// SIMATIC S7-200 project (STEP 7-Micro/WIN), CPU 224XP REL 02.01

SYMBOL_TABLE USER1
P0               M0.0
END_SYMBOL_TABLE

ORGANIZATION_BLOCK MAIN:OB1
TITLE=PROGRAM COMMENTS
BEGIN
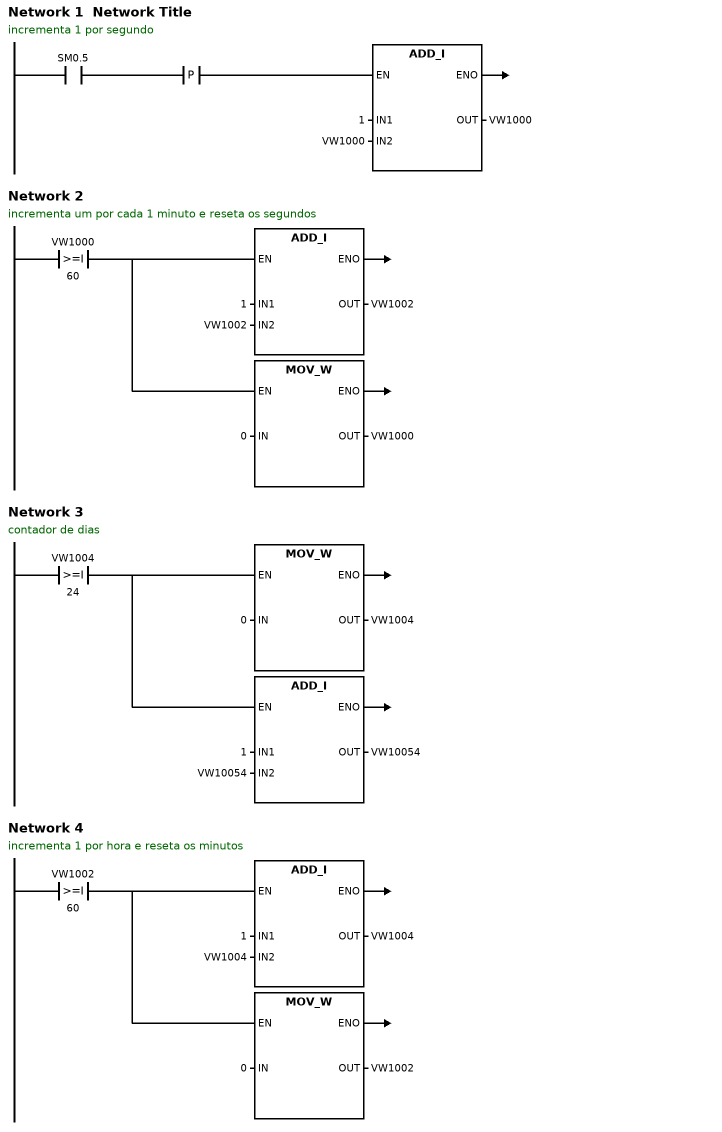
Network 1 // Network Title
// incrementa 1 por segundo
LD     SM0.5
EU
+I     1, VW1000
Network 2
// incrementa um por cada 1 minuto e reseta os segundos
LDW>=  VW1000, 60
+I     1, VW1002
MOVW   0, VW1000
Network 3
// contador de dias
LDW>=  VW1004, 24
MOVW   0, VW1004
+I     1, VW10054
Network 4
// incrementa 1 por hora e reseta os minutos
LDW>=  VW1002, 60
+I     1, VW1004
MOVW   0, VW1002
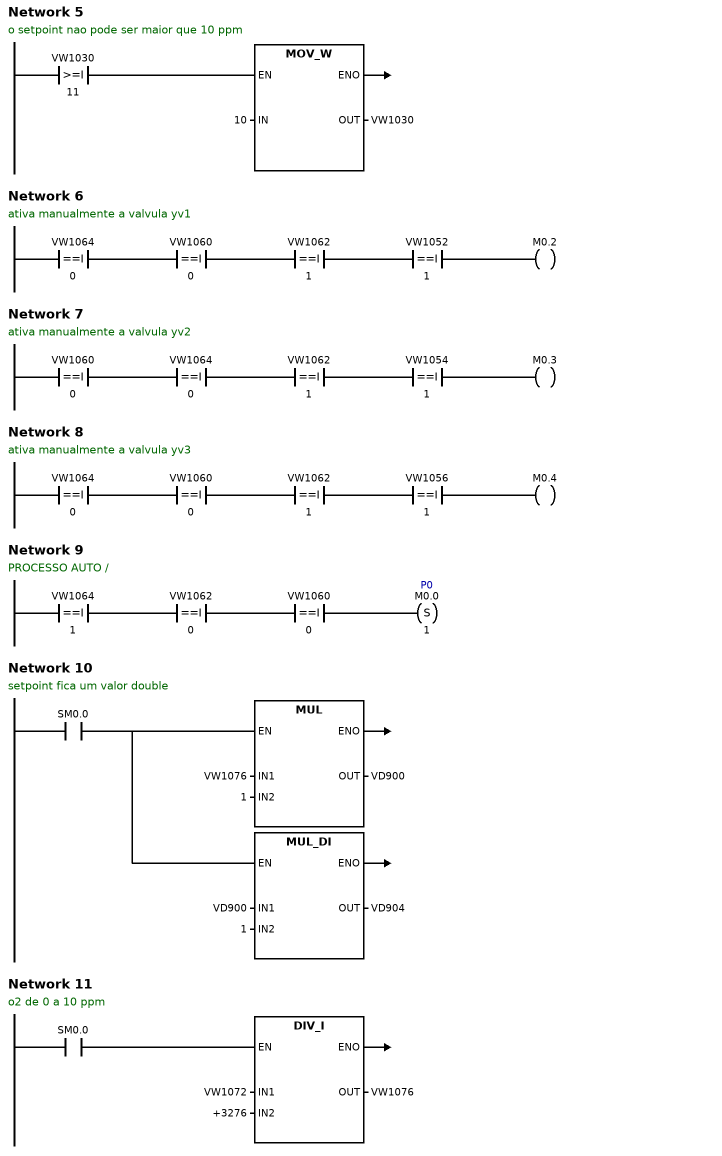
Network 5
// o setpoint nao pode ser maior que 10 ppm
LDW>=  VW1030, 11
MOVW   10, VW1030
Network 6
// ativa manualmente a valvula yv1
LDW=   VW1064, 0
AW=    VW1060, 0
AW=    VW1062, 1
AW=    VW1052, 1
=      M0.2
Network 7
// ativa manualmente a valvula yv2
LDW=   VW1060, 0
AW=    VW1064, 0
AW=    VW1062, 1
AW=    VW1054, 1
=      M0.3
Network 8
// ativa manualmente a valvula yv3
LDW=   VW1064, 0
AW=    VW1060, 0
AW=    VW1062, 1
AW=    VW1056, 1
=      M0.4
Network 9
// PROCESSO AUTO
// 
LDW=   VW1064, 1
AW=    VW1062, 0
AW=    VW1060, 0
S      P0:M0.0, 1
Network 10
// setpoint fica um valor double
LD     SM0.0
MOVW   VW1076, VW902
MUL    1, VD900
MOVD   VD900, VD904
*D     1, VD904
Network 11
// o2 de 0 a 10 ppm
LD     SM0.0
MOVW   VW1072, VW1076
/I     +3276, VW1076
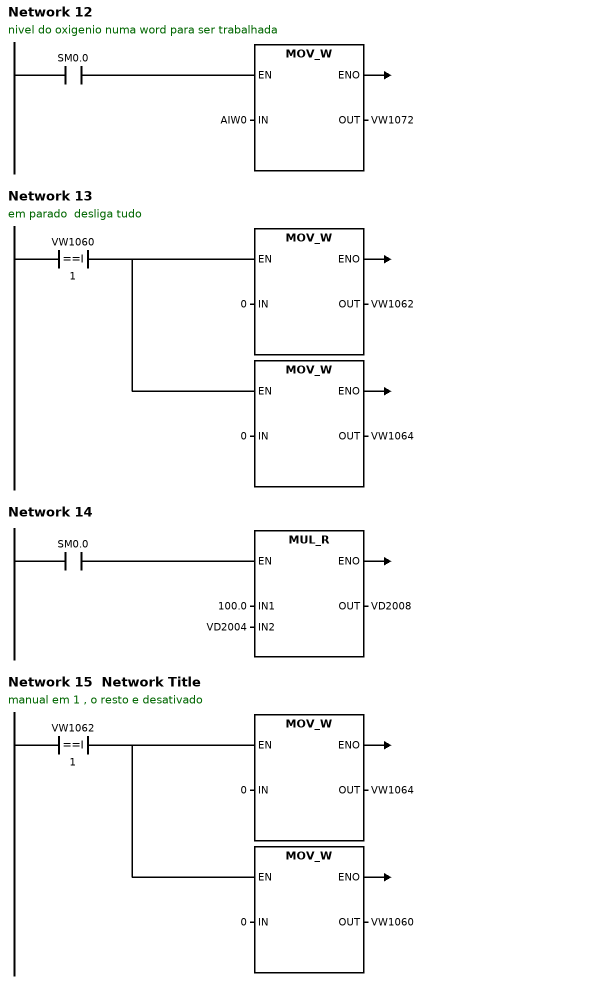
Network 12
// nivel do oxigenio numa word para ser trabalhada 
LD     SM0.0
MOVW   AIW0, VW1072
Network 13
// em parado  desliga tudo
LDW=   VW1060, 1
MOVW   0, VW1062
MOVW   0, VW1064
Network 14
LD     SM0.0
MOVR   100.0, VD2008
*R     VD2004, VD2008
Network 15 // Network Title
// manual em 1 , o resto e desativado
LDW=   VW1062, 1
MOVW   0, VW1064
MOVW   0, VW1060
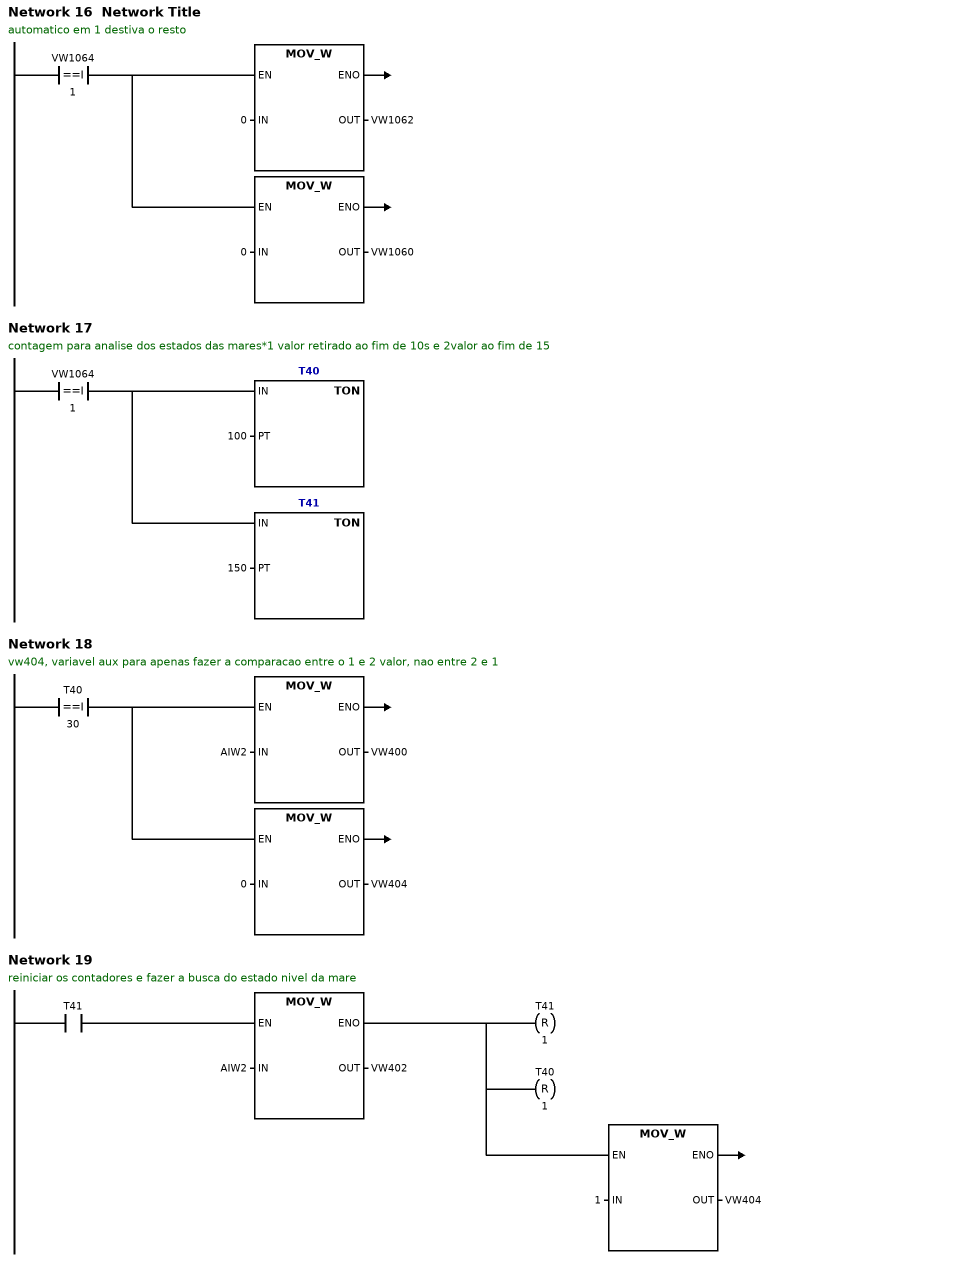
Network 16 // Network Title
// automatico em 1 destiva o resto
LDW=   VW1064, 1
MOVW   0, VW1062
MOVW   0, VW1060
Network 17
// contagem para analise dos estados das mares*1 valor retirado ao fim de 10s e 2valor ao fim de 15
LDW=   VW1064, 1
TON    T40, 100
TON    T41, 150
Network 18
// vw404, variavel aux para apenas fazer a comparacao entre o 1 e 2 valor, nao entre 2 e 1
LDW=   T40, 30
MOVW   AIW2, VW400
MOVW   0, VW404
Network 19
// reiniciar os contadores e fazer a busca do estado nivel da mare
LD     T41
MOVW   AIW2, VW402
AENO
R      T41, 1
R      T40, 1
MOVW   1, VW404
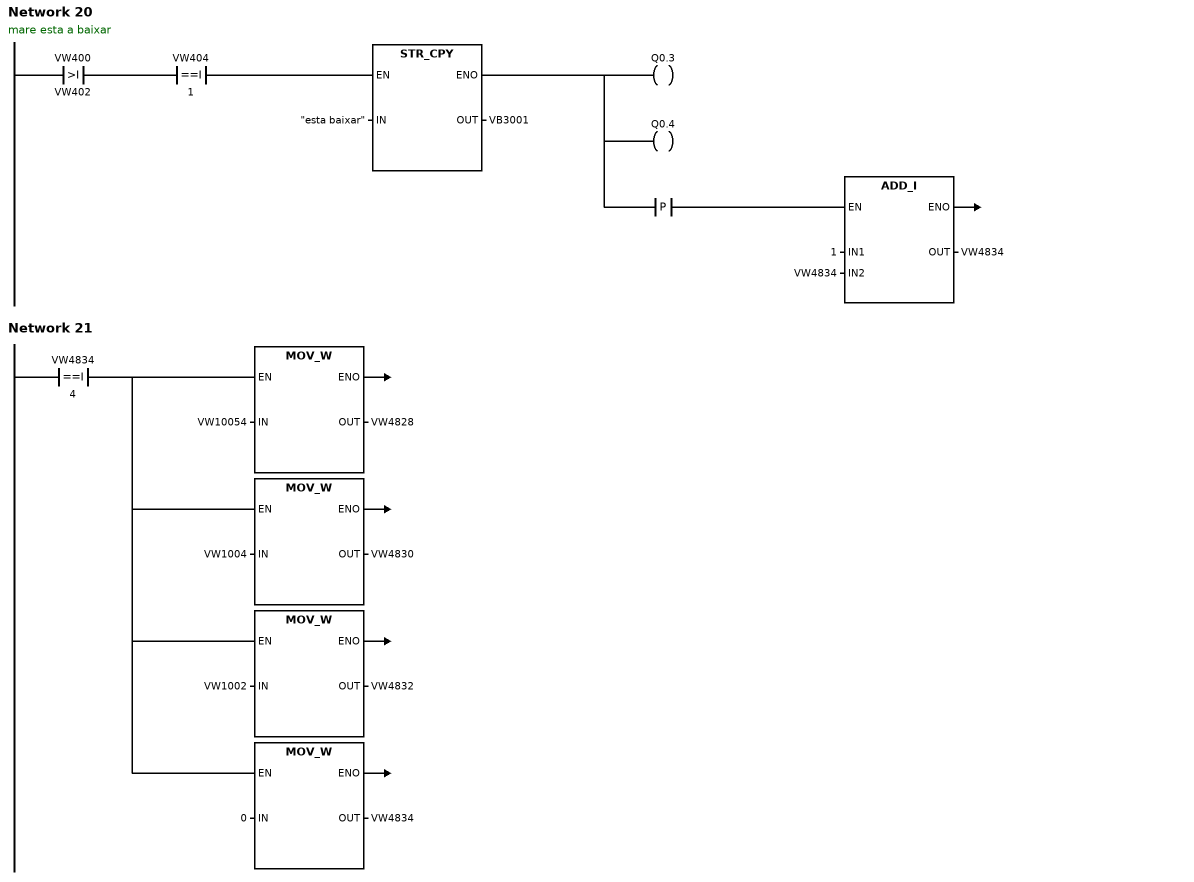
Network 20
// mare esta a baixar
LDW>   VW400, VW402
AW=    VW404, 1
SCPY   "esta baixar", VB3001
AENO
=      Q0.3
=      Q0.4
EU
+I     1, VW4834
Network 21
LDW=   VW4834, 4
MOVW   VW10054, VW4828
MOVW   VW1004, VW4830
MOVW   VW1002, VW4832
MOVW   0, VW4834
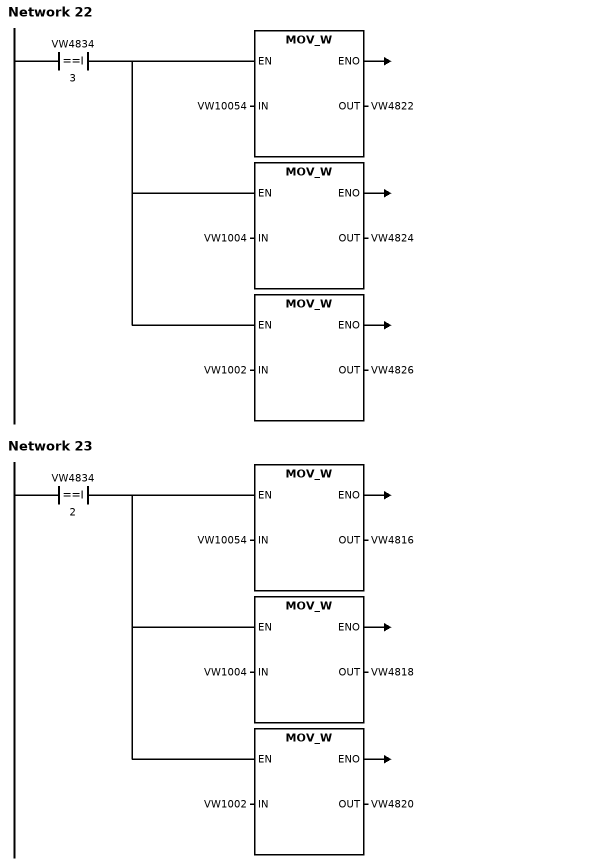
Network 22
LDW=   VW4834, 3
MOVW   VW10054, VW4822
MOVW   VW1004, VW4824
MOVW   VW1002, VW4826
Network 23
LDW=   VW4834, 2
MOVW   VW10054, VW4816
MOVW   VW1004, VW4818
MOVW   VW1002, VW4820
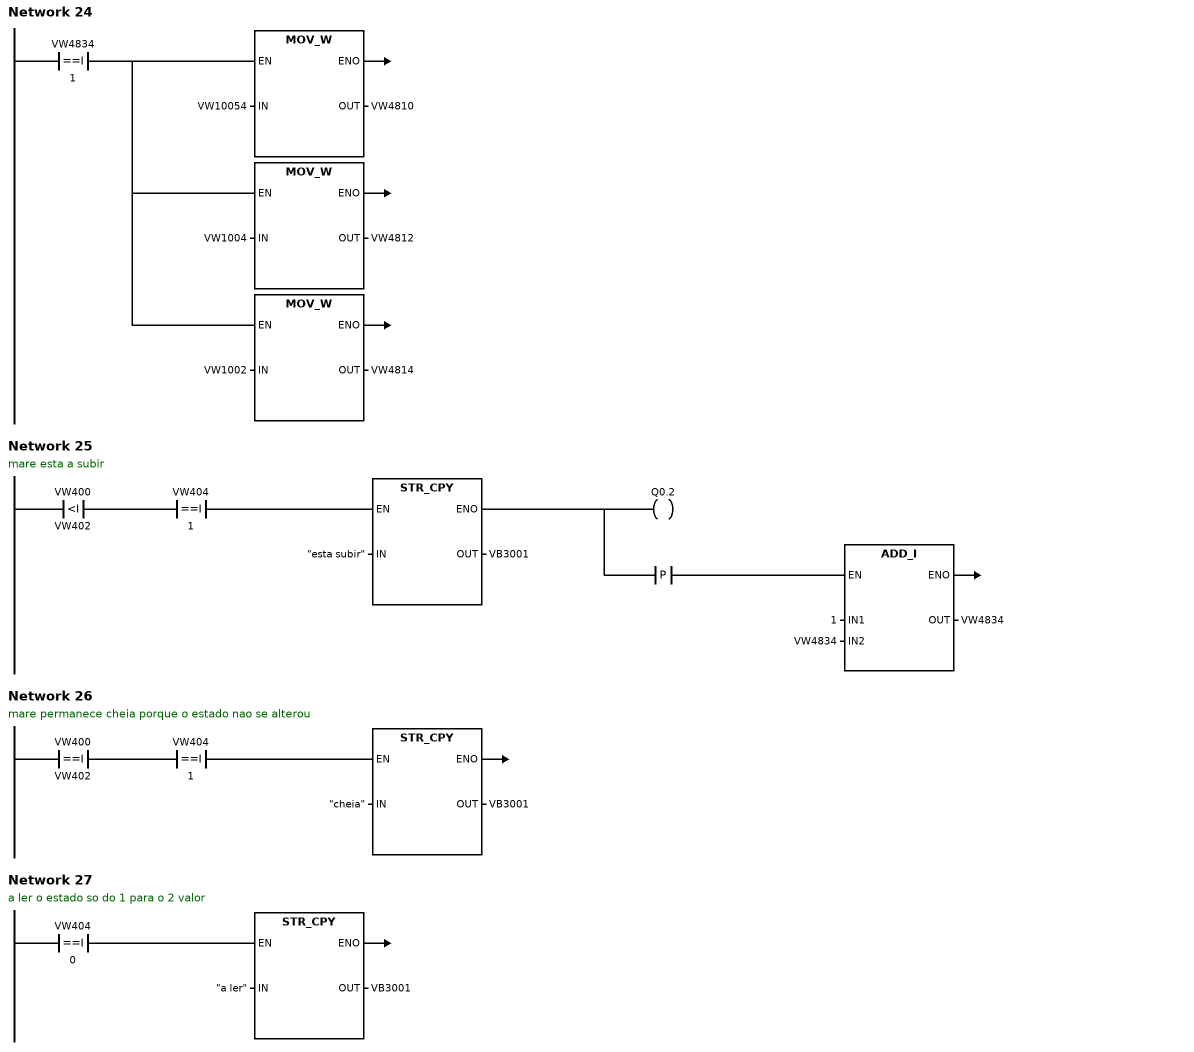
Network 24
LDW=   VW4834, 1
MOVW   VW10054, VW4810
MOVW   VW1004, VW4812
MOVW   VW1002, VW4814
Network 25
// mare esta a subir
LDW<   VW400, VW402
AW=    VW404, 1
SCPY   "esta subir", VB3001
AENO
=      Q0.2
EU
+I     1, VW4834
Network 26
// mare permanece cheia porque o estado nao se alterou
LDW=   VW400, VW402
AW=    VW404, 1
SCPY   "cheia", VB3001
Network 27
// a ler o estado so do 1 para o 2 valor
LDW=   VW404, 0
SCPY   "a ler", VB3001
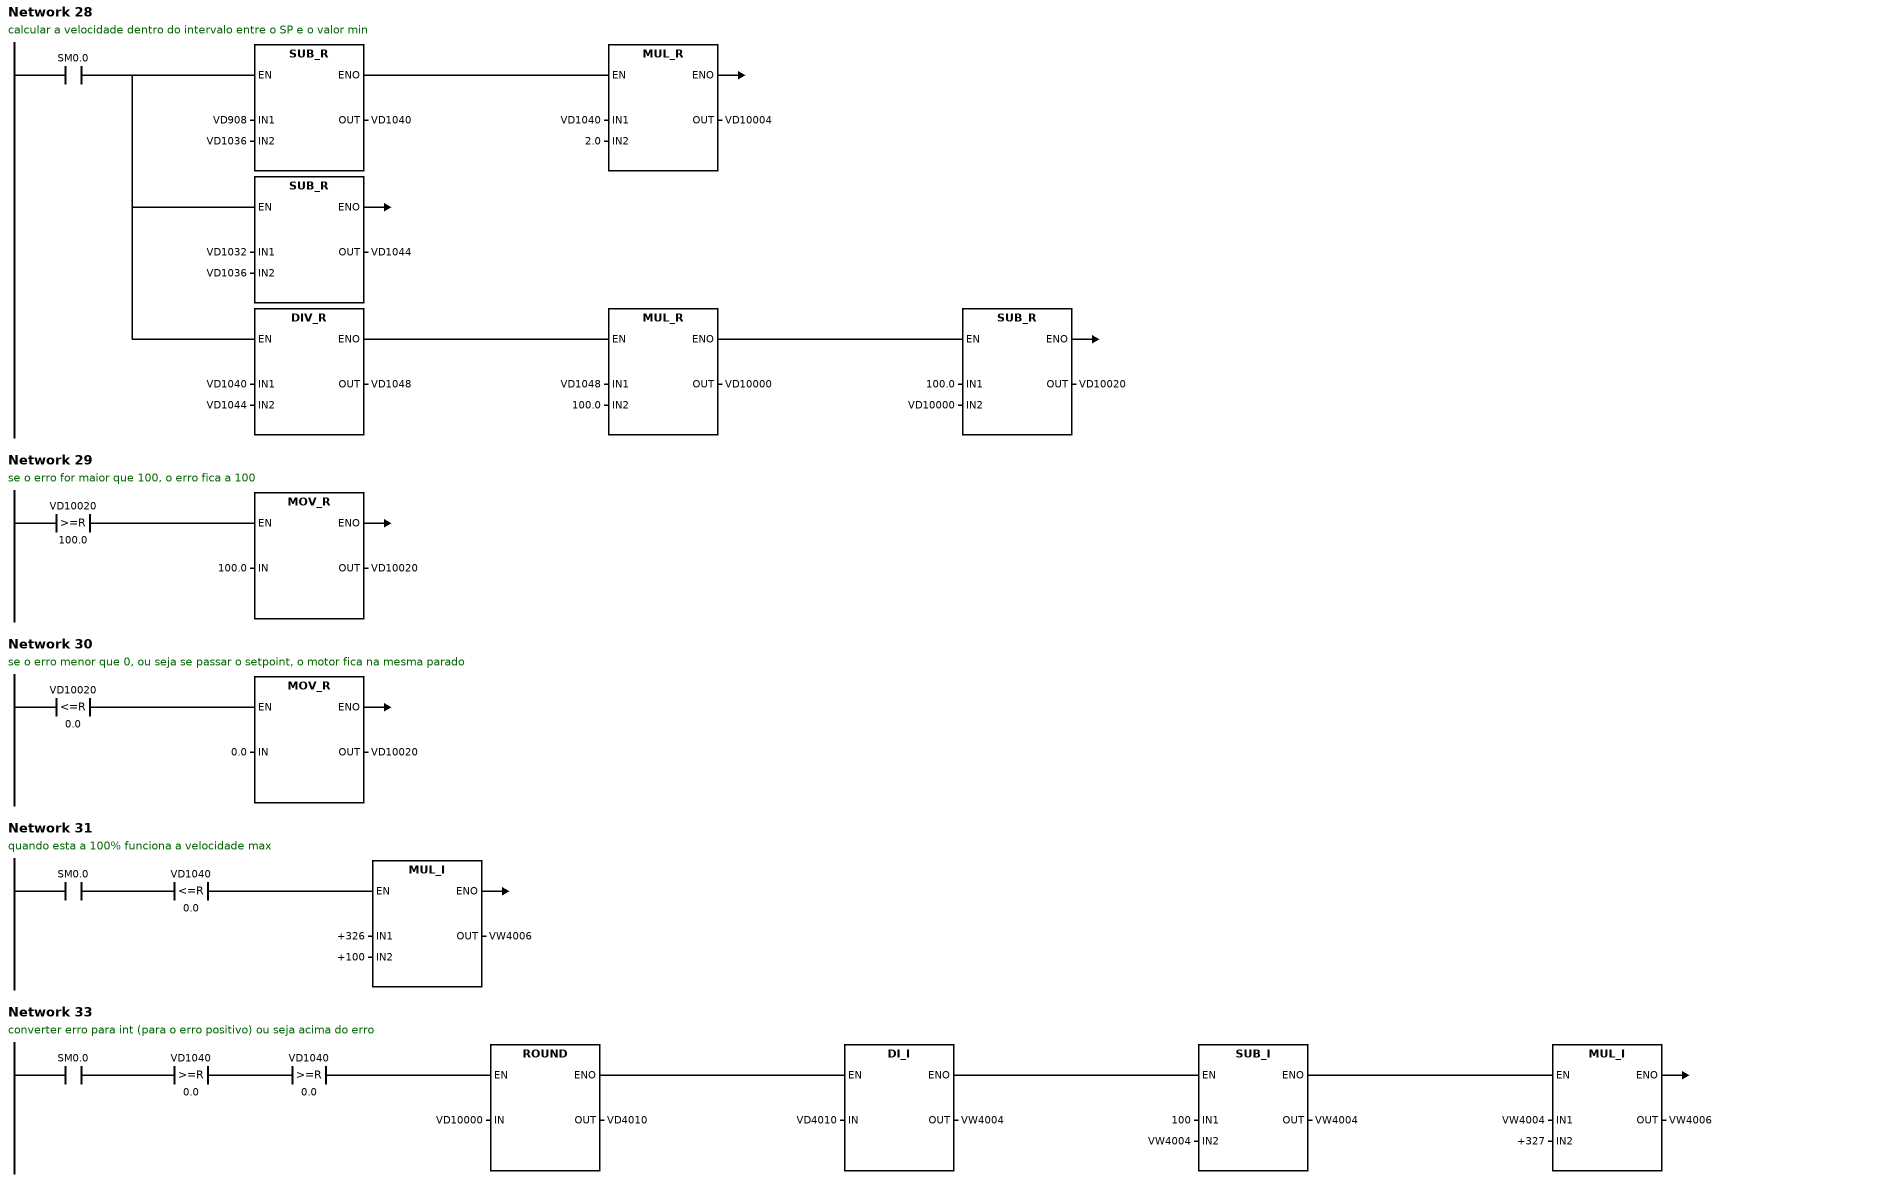
Network 28
// calcular a velocidade dentro do intervalo entre o SP e o valor min
LD     SM0.0
LPS
MOVR   VD908, VD1040
AENO
-R     VD1036, VD1040
AENO
MOVR   VD1040, VD10004
*R     2.0, VD10004
LRD
MOVR   VD1032, VD1044
-R     VD1036, VD1044
LPP
MOVR   VD1040, VD1048
AENO
/R     VD1044, VD1048
AENO
MOVR   VD1048, VD10000
AENO
*R     100.0, VD10000
AENO
MOVR   100.0, VD10020
-R     VD10000, VD10020
Network 29
// se o erro for maior que 100, o erro fica a 100
LDR>=  VD10020, 100.0
MOVR   100.0, VD10020
Network 30
// se o erro menor que 0, ou seja se passar o setpoint, o motor fica na mesma parado
LDR<=  VD10020, 0.0
MOVR   0.0, VD10020
Network 31
// quando esta a 100% funciona a velocidade max
LD     SM0.0
AR<=   VD1040, 0.0
MOVW   +326, VW4006
*I     +100, VW4006
Network 33
// converter erro para int (para o erro positivo) ou seja acima do erro
LD     SM0.0
AR>=   VD1040, 0.0
AR>=   VD1040, 0.0
ROUND  VD10000, VD4010
AENO
DTI    VD4010, VW4004
AENO
INVW   VW4004
AENO
INCW   VW4004
AENO
+I     100, VW4004
AENO
MOVW   VW4004, VW4006
*I     +327, VW4006
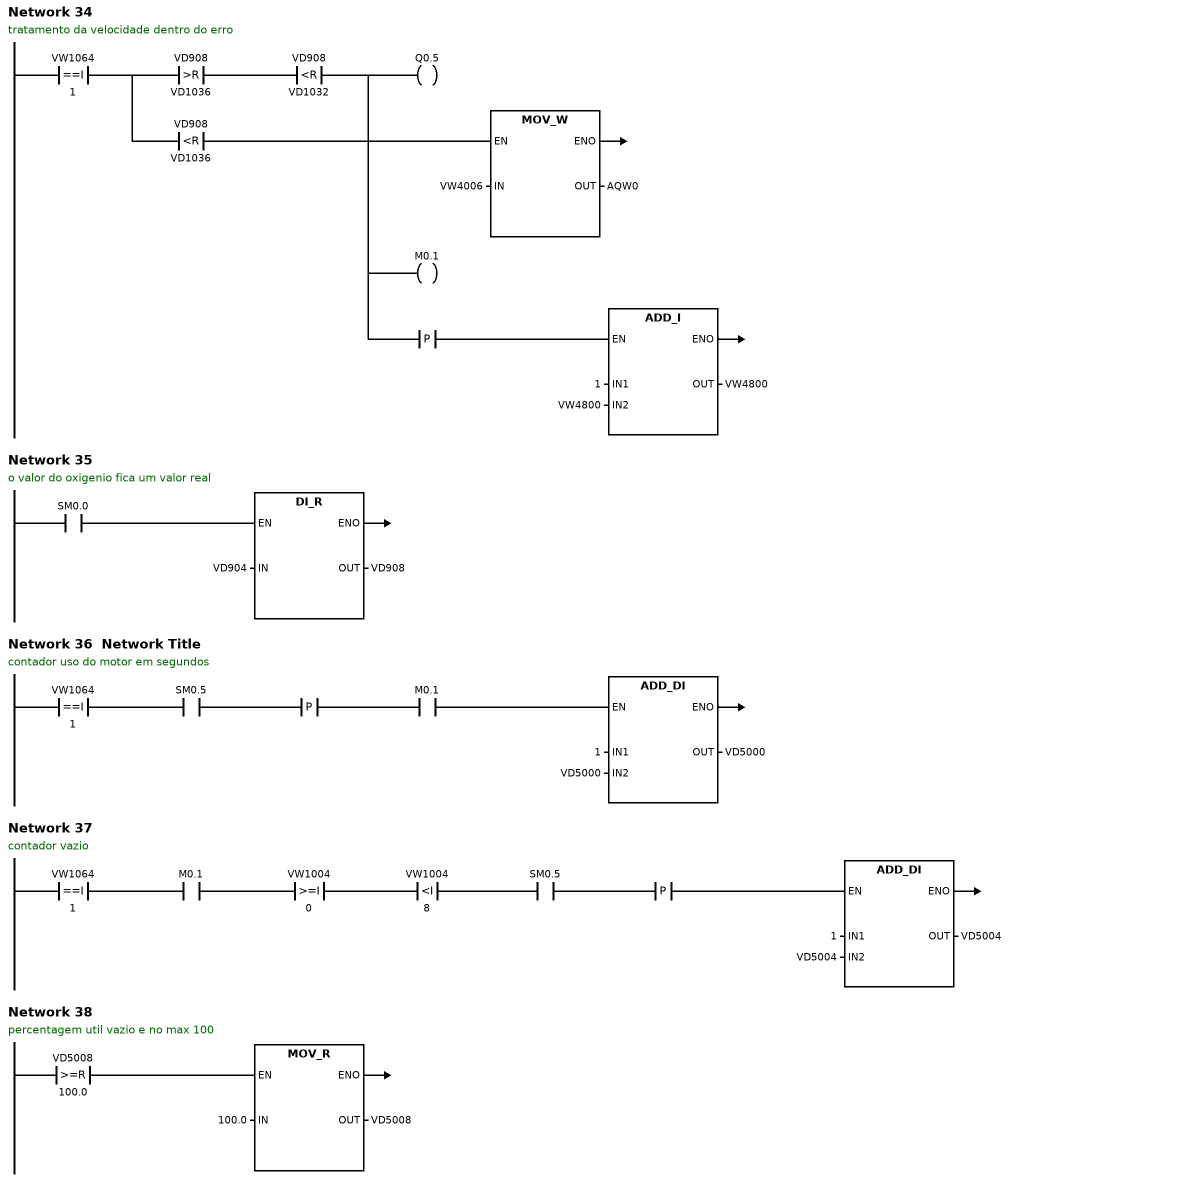
Network 34
// tratamento da velocidade dentro do erro
LDW=   VW1064, 1
LDR>   VD908, VD1036
AR<    VD908, VD1032
OR<    VD908, VD1036
ALD
=      Q0.5
MOVW   VW4006, AQW0
=      M0.1
EU
+I     1, VW4800
Network 35
// o valor do oxigenio fica um valor real
LD     SM0.0
DTR    VD904, VD908
Network 36 // Network Title
// contador uso do motor em segundos 
LDW=   VW1064, 1
A      SM0.5
EU
A      M0.1
+D     1, VD5000
Network 37
// contador vazio
LDW=   VW1064, 1
A      M0.1
AW>=   VW1004, 0
AW<    VW1004, 8
A      SM0.5
EU
+D     1, VD5004
Network 38
// percentagem util vazio e no max 100 
LDR>=  VD5008, 100.0
MOVR   100.0, VD5008
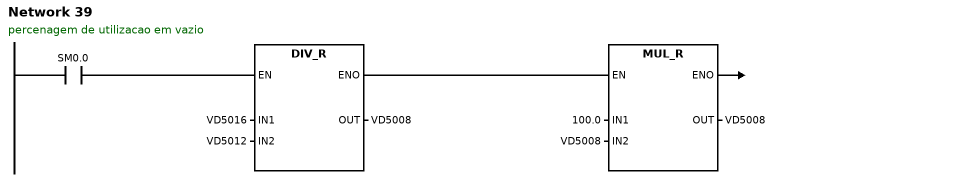
Network 39
// percenagem de utilizacao em vazio
LD     SM0.0
MOVR   VD5016, VD5008
AENO
/R     VD5012, VD5008
AENO
*R     100.0, VD5008
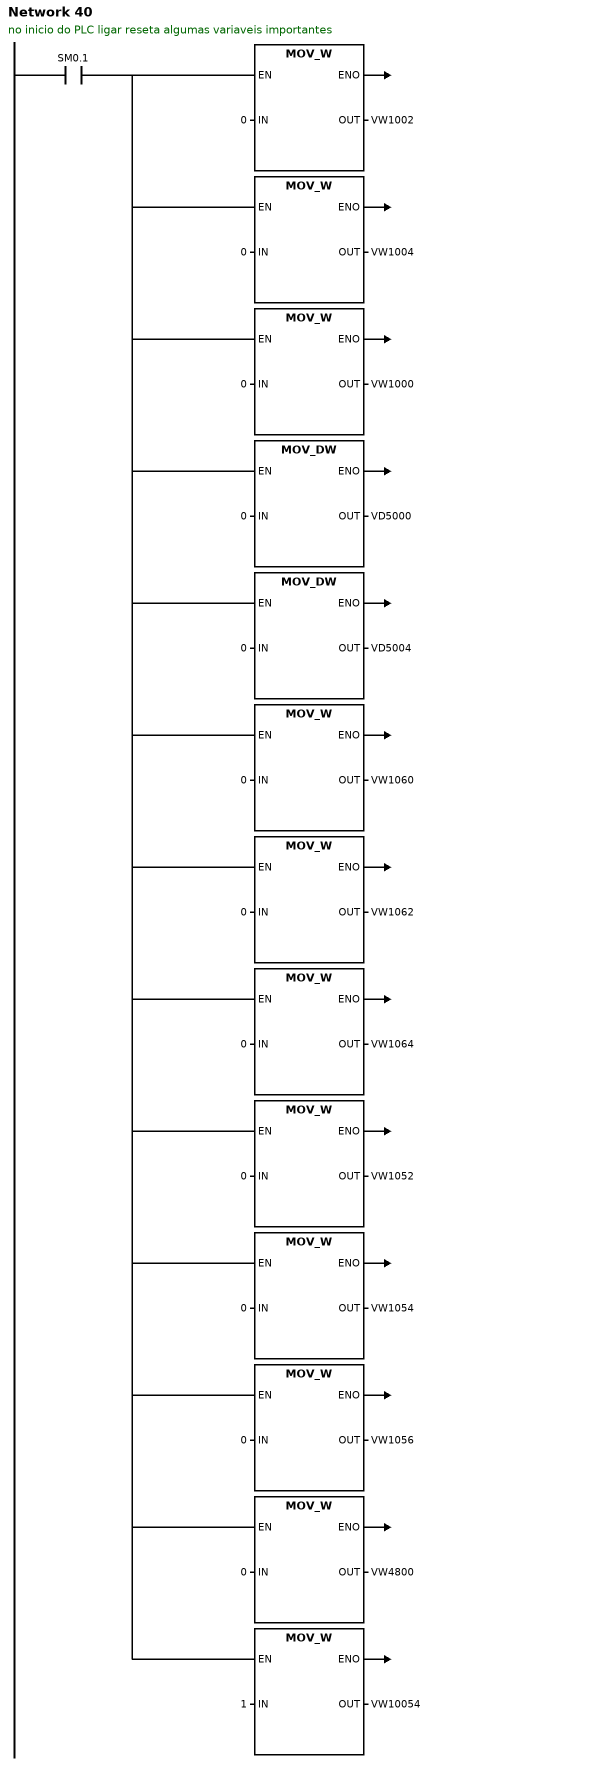
Network 40
// no inicio do PLC ligar reseta algumas variaveis importantes
LD     SM0.1
MOVW   0, VW1002
MOVW   0, VW1004
MOVW   0, VW1000
MOVD   0, VD5000
MOVD   0, VD5004
MOVW   0, VW1060
MOVW   0, VW1062
MOVW   0, VW1064
MOVW   0, VW1052
MOVW   0, VW1054
MOVW   0, VW1056
MOVW   0, VW4800
MOVW   1, VW10054
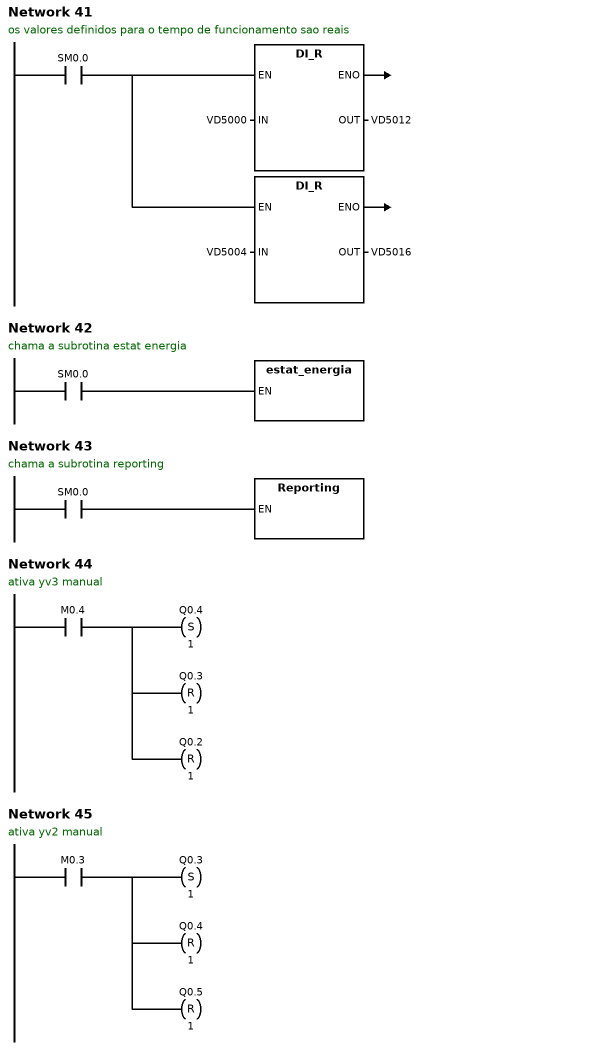
Network 41
// os valores definidos para o tempo de funcionamento sao reais
LD     SM0.0
DTR    VD5000, VD5012
DTR    VD5004, VD5016
Network 42
// chama a subrotina estat energia
LD     SM0.0
CALL   estat_energia:SBR0
Network 43
// chama a subrotina reporting
LD     SM0.0
CALL   Reporting:SBR3
Network 44
// ativa yv3 manual
LD     M0.4
S      Q0.4, 1
R      Q0.3, 1
R      Q0.2, 1
Network 45
// ativa yv2 manual
LD     M0.3
S      Q0.3, 1
R      Q0.4, 1
R      Q0.5, 1
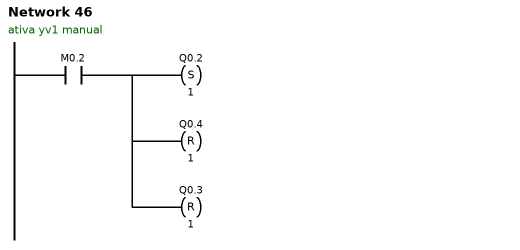
Network 46
// ativa yv1 manual
LD     M0.2
S      Q0.2, 1
R      Q0.4, 1
R      Q0.3, 1
END_ORGANIZATION_BLOCK

SUBROUTINE_BLOCK estat_energia:SBR0
TITLE=SUBROUTINE COMMENTS
BEGIN
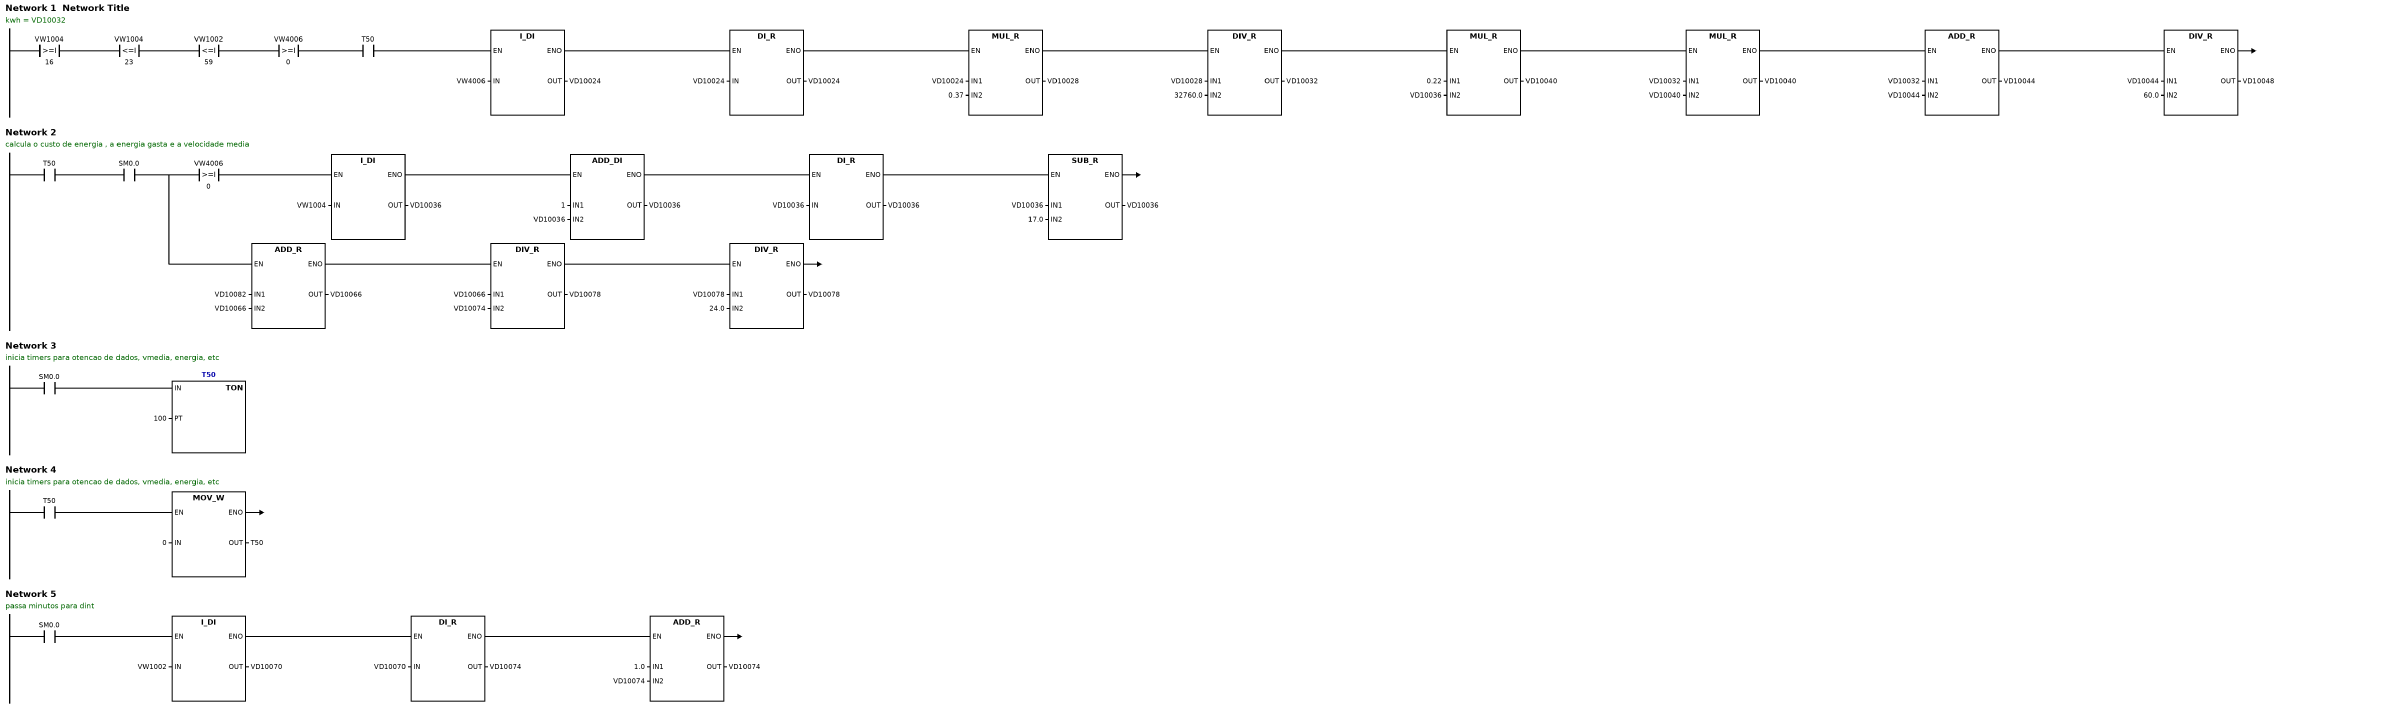
Network 1 // Network Title
// kwh = VD10032
LDW>=  VW1004, 16
AW<=   VW1004, 23
AW<=   VW1002, 59
AW>=   VW4006, 0
A      T50
ITD    VW4006, VD10024
AENO
DTR    VD10024, VD10024
AENO
MOVR   VD10024, VD10028
AENO
*R     0.37, VD10028
AENO
MOVR   VD10028, VD10032
AENO
/R     32760.0, VD10032
AENO
MOVR   0.22, VD10040
AENO
*R     VD10036, VD10040
AENO
*R     VD10032, VD10040
AENO
+R     VD10032, VD10044
AENO
MOVR   VD10044, VD10048
/R     60.0, VD10048
Network 2
// calcula o custo de energia , a energia gasta e a velocidade media 
LD     T50
A      SM0.0
LPS
AW>=   VW4006, 0
ITD    VW1004, VD10036
AENO
+D     1, VD10036
AENO
DTR    VD10036, VD10036
AENO
-R     17.0, VD10036
LPP
+R     VD10082, VD10066
AENO
MOVR   VD10066, VD10078
AENO
/R     VD10074, VD10078
AENO
/R     24.0, VD10078
Network 3
// inicia timers para otencao de dados, vmedia, energia, etc
LD     SM0.0
TON    T50, 100
Network 4
// inicia timers para otencao de dados, vmedia, energia, etc
LD     T50
MOVW   0, T50
Network 5
// passa minutos para dint
LD     SM0.0
ITD    VW1002, VD10070
AENO
DTR    VD10070, VD10074
AENO
+R     1.0, VD10074
END_SUBROUTINE_BLOCK

// SBR1: protected block, not included

// SBR2: protected block, not included

SUBROUTINE_BLOCK Reporting:SBR3
TITLE=SUBROUTINE COMMENTS
BEGIN
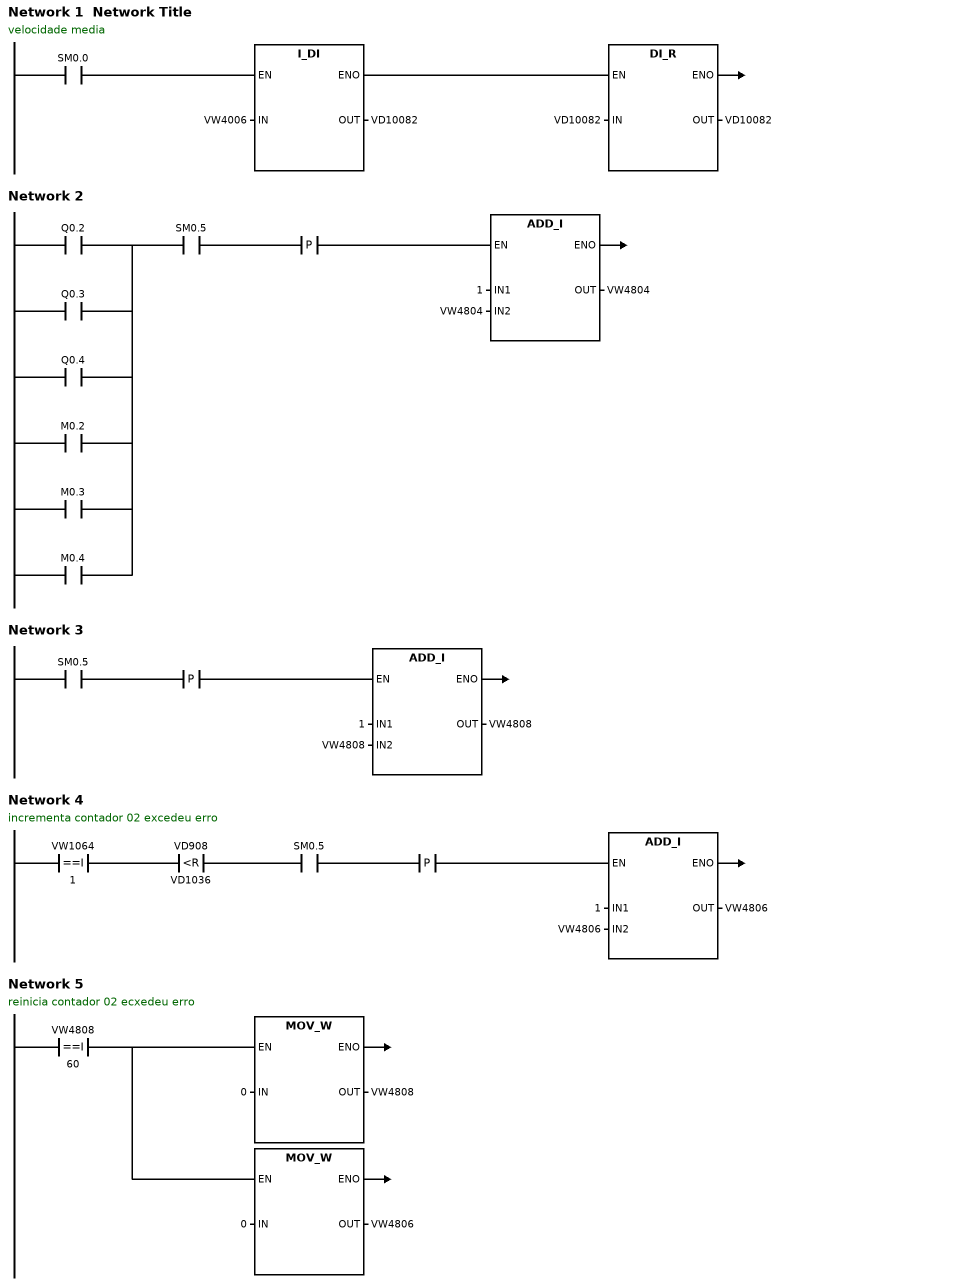
Network 1 // Network Title
// velocidade media
LD     SM0.0
ITD    VW4006, VD10082
AENO
DTR    VD10082, VD10082
Network 2
LD     Q0.2
O      Q0.3
O      Q0.4
O      M0.2
O      M0.3
O      M0.4
A      SM0.5
EU
+I     1, VW4804
Network 3
LD     SM0.5
EU
+I     1, VW4808
Network 4
// incrementa contador 02 excedeu erro
LDW=   VW1064, 1
AR<    VD908, VD1036
A      SM0.5
EU
+I     1, VW4806
Network 5
// reinicia contador 02 ecxedeu erro
LDW=   VW4808, 60
MOVW   0, VW4808
MOVW   0, VW4806
END_SUBROUTINE_BLOCK

// (further data pages could not be read)
